// TIA Portal V20 export
VAR_GLOBAL   // PLC tag table "PHMI"
   "BA010AZCRD1PHMI.I[0]" AT %IW6 : Int;   //    {ExternalVisible false}
   "BA010AZCRD1PHMI.Q[0]" AT %QW6 : Int;   //    {ExternalVisible false}
END_VAR
